(* IEC 61131-3 sources: eCockpitGit/test_project/src/%F%03 Module/%POU%FB_Module/%F%Action/%PRO%hasAction, 1 file *)

(* ---- %GETSET%Get.st ---- *)
VAR
END_VAR

(*%!%__DELIMITER__%!%*)
hasAction		:=		FALSE;
